(* IEC 61131-3 sources: types/src (part 3) *)

   END_TYPE

   TYPE EM480VHFDataRec145V1 : STRUCT
         version  : Byte := BYTE#1;   // Version
         resb1  : Byte;   // Reserved
         minVoltL1N  : Real;   // Min. voltage UL1-N
         minVoltL2N  : Real;   // Min. voltage UL2-N
         minVoltL3N  : Real;   // Min. voltage UL3-N
         minVoltL1L2  : Real;   // Min. voltage UL1-L2
         minVoltL2L3  : Real;   // Min. voltage UL2-L3
         minVoltL3L1  : Real;   // Min. voltage UL3-L1
         minCurrentL1  : Real;   // Min. current L1
         minCurrentL2  : Real;   // Min. current L2
         minCurrentL3  : Real;   // Min. current L3
         minApparentPowerL1  : Real;   // Min. apparent power L1
         minApparentPowerL2  : Real;   // Min. apparent power L2
         minApparentPowerL3  : Real;   // Min. apparent power L3
         minActivePowerL1  : Real;   // Min. active power L1
         minActivePowerL2  : Real;   // Min. active power L2
         minActivePowerL3  : Real;   // Min. active power L3
         minReactivePowerQtotL1  : Real;   // Min. reactive power Qtot L1
         minReactivePowerQtotL2  : Real;   // Min. reactive power Qtot L2
         minReactivePowerQtotL3  : Real;   // Min. reactive power Qtot L3
         minPowerFactorL1  : Real;   // Min. power factor L1
         minPowerFactorL2  : Real;   // Min. power factor L2
         minPowerFactorL3  : Real;   // Min. power factor L3
         minFrequency  : Real;   // Min. frequency
         minTotalApparentPower  : Real;   // Min. apparent power L1 L2 L3
         minTotalActivePower  : Real;   // Min. active power L1 L2 L3
         minTotalReactivePowerQn  : Real;   // Min. reactive power Qn L1 L2 L3
         minTotalPowerFactor  : Real;   // Min. power factor λ L1 L2 L3
         minReactivePowerQnL1  : Real;   // Min. reactive power Qn L1
         minReactivePowerQnL2  : Real;   // Min. reactive power Qn L2
         minReactivePowerQnL3  : Real;   // Min. reactive power Qn L3
         minMeanVoltLN  : Real;   // Min. mean voltage L-N
         minMeanVoltLL  : Real;   // Min. mean voltage L-L
         minTotalMeanCurr  : Real;   // Min. mean current L1 L2 L3
         minFundVoltL1  : Real;   // Min. fundamental voltage L1
         minFundVoltL2  : Real;   // Min. fundamental voltage L2
         minFundVoltL3  : Real;   // Min. fundamental voltage L3
         minFundCurrL1  : Real;   // Min. fundamental current L1
         minFundCurrL2  : Real;   // Min. fundamental current L2
         minFundCurrL3  : Real;   // Min. fundamental current L3
         minFundApparentPowerL1  : Real;   // Min. fundamental apparent power L1
         minFundApparentPowerL2  : Real;   // Min. fundamental apparent power L2
         minFundApparentPowerL3  : Real;   // Min. fundamental apparent power L3
         minFundReactivePowerL1  : Real;   // Min. fundamental reactive power L1
         minFundReactivePowerL2  : Real;   // Min. fundamental reactive power L2
         minFundReactivePowerL3  : Real;   // Min. fundamental reactive power L3
         minFundActivePowerL1  : Real;   // Min. fundamental active power L1
         minFundActivePowerL2  : Real;   // Min. fundamental active power L2
         minFundActivePowerL3  : Real;   // Min. fundamental active power L3
         minFundActiveFactorL1  : Real;   // Min. fundamental cos φ active factor L1
         minFundActiveFactorL2  : Real;   // Min. fundamental cos φ active factor L2
         minFundActiveFactorL3  : Real;   // Min. fundamental cos φ active factor L3
         minTHDaNVoltL1  : Real;   // Min. THD+N voltage L1
         minTHDaNVoltL2  : Real;   // Min. THD+N voltage L2
         minTHDaNVoltL3  : Real;   // Min. THD+N voltage L3
         minTHDaNCurrL1  : Real;   // Min. THD+N current L1
         minTHDaNCurrL2  : Real;   // Min. THD+N current L2
         minTHDaNCurrL3  : Real;   // Min. THD+N current L3
      END_STRUCT;

   END_TYPE

   TYPE EM480VHFDataRec143 : STRUCT
         version  : Byte := BYTE#1;   // Version
         resb1  : Byte;   // Reserved
         controlStatusByte1L1  : Byte;   // Status / control byte 1 - L1
         controlStatusByte2L1  : Byte;   // Status / control byte 2 - L1
         controlStatusByte1L2  : Byte;   // Status / control byte 1 - L2
         controlStatusByte2L2  : Byte;   // Status / control byte 2 - L2
         controlStatusByte1L3  : Byte;   // Status / control byte 1 - L3
         controlStatusByte2L3  : Byte;   // Status / control byte 2 - L3
         activeEnergyInLongL1  : LReal;   // Active energy inflow (initial value) L1
         activeEnergyOutLongL1  : LReal;   // Active energy outflow (initial value) L1
         reactiveEnergyInLongL1  : LReal;   // Reactive energy inflow (initial value) L1
         reactiveEnergyOutLongL1  : LReal;   // Reactive energy outflow (initial value) L1
         apparentEnergyLongL1  : LReal;   // Apparent energy (initial value) L1
         activeEnergyInLongL2  : LReal;   // Active energy inflow (initial value) L2
         activeEnergyOutLongL2  : LReal;   // Active energy outflow (initial value) L2
         reactiveEnergyInLongL2  : LReal;   // Reactive energy inflow (initial value) L2
         reactiveEnergyOutLongL2  : LReal;   // Reactive energy outflow (initial value) L2
         apparentEnergyLongL2  : LReal;   // Apparent energy (initial value) L2
         activeEnergyInLongL3  : LReal;   // Active energy inflow (initial value) L3
         activeEnergyOutLongL3  : LReal;   // Active energy outflow (initial value) L3
         reactiveEnergyInLongL3  : LReal;   // Reactive energy inflow (initial value) L3
         reactiveEnergyOutLongL3  : LReal;   // Reactive energy outflow (initial value) L3
         apparentEnergyLongL3  : LReal;   // Apparent energy (initial value) L3
         ovCntActiveEnergyInL1  : UInt;   // Overflow counter active energy inflow L1
         ovCntActiveEnergyOutL1  : UInt;   // Overflow counter active energy outflow L1
         ovCntReactiveEnergyInL1  : UInt;   // Overflow counter reactive energy inflow L1
         ovCntReactiveEnergyOutL1  : UInt;   // Overflow counter reactive energy outflow L1
         ovCntApparentEnergyL1  : UInt;   // Overflow counter apparent energy L1
         ovCntActiveEnergyInL2  : UInt;   // Overflow counter active energy inflow L2
         ovCntActiveEnergyOutL2  : UInt;   // Overflow counter active energy outflow L2
         ovCntReactiveEnergyInL2  : UInt;   // Overflow counter reactive energy inflow L2
         ovCntReactiveEnergyOutL2  : UInt;   // Overflow counter reactive energy outflow L2
         ovCntApparentEnergyL2  : UInt;   // Overflow counter apparent energy L2
         ovCntActiveEnergyInL3  : UInt;   // Overflow counter active energy inflow L3
         ovCntActiveEnergyOutL3  : UInt;   // Overflow counter active energy outflow L3
         ovCntReactiveEnergyInL3  : UInt;   // Overflow counter reactive energy inflow L3
         ovCntReactiveEnergyOutL3  : UInt;   // Overflow counter reactive energy outflow L3
         ovCntApparentEnergyL3  : UInt;   // Overflow counter apparent energy L3
         operHoursCntL1  : Real;   // Operating hours counter L1 (initial value)
         operHoursCntL2  : Real;   // Operating hours counter L2 (initial value)
         operHoursCntL3  : Real;   // Operating hours counter L2 (initial value)
      END_STRUCT;

   END_TYPE

   TYPE EM480VHFDataRec142V2 : STRUCT
         version  : Byte := BYTE#2;   // Version
         resb1  : Byte;   // Reserved
         voltL1N  : Real;   // Voltage UL1-N
         voltL2N  : Real;   // Voltage UL2-N
         voltL3N  : Real;   // Voltage UL3-N
         voltL1L2  : Real;   // Voltage UL1-L2
         voltL2L3  : Real;   // Voltage UL2-L3
         voltL3L1  : Real;   // Voltage UL3-L1
         currentL1  : Real;   // Current L1
         currentL2  : Real;   // Current L2
         currentL3  : Real;   // Current L3
         powerFactorL1  : Real;   // Power factor L1
         powerFactorL2  : Real;   // Power factor L2
         powerFactorL3  : Real;   // Power factor L3
         totalPowerFactor  : Real;   // Total power factor L1 L2 L3
         frequency  : Real;   // Frequency
         amplUnbalanceVolt  : Real;   // Amplitude unbalance for voltage
         amplUnbalanceCurrent  : Real;   // Amplitude unbalance for current
         apparentPowerL1  : Real;   // Apparent power L1
         apparentPowerL2  : Real;   // Apparent power L2
         apparentPowerL3  : Real;   // Apparent power L3
         totalApparentPower  : Real;   // Total apparent power L1 L2 L3
         reactivePowerQtotL1  : Real;   // Reactive power Qtot L1
         reactivePowerQtotL2  : Real;   // Reactive power Qtot L2
         reactivePowerQtotL3  : Real;   // Reactive power Qtot L2
         totalReactivePowerQtot  : Real;   // Total reactive power Qtot L1 L2 L3
         activePowerL1  : Real;   // Active power L1
         activePowerL2  : Real;   // Active power L2
         activePowerL3  : Real;   // Active power L3
         totalActivePower  : Real;   // Total active power L1 L2 L3
         phaseAngleL1  : Real;   //  Phase angle L1
         phaseAngleL2  : Real;   //  Phase angle L2
         phaseAngleL3  : Real;   //  Phase angle L3
         totalApparentEnergy  : Real;   // Total apparent energy L1 L2 L3
         totalReactiveEnergy  : Real;   // Total reactive energy L1 L2 L3
         totalActiveEnergy  : Real;   // Total active energy L1 L2 L3
         totalReactiveEnergyIn  : Real;   // Total reactive energy inflow L1 L2 L3
         totalReactiveEnergyOut  : Real;   // Total reactive energy outflow L1 L2 L3
         totalActiveEnergyIn  : Real;   // Total active energy inflow L1 L2 L3
         totalActiveEnergyOut  : Real;   // Total active energy outflow L1 L2 L3
         totalApparentEnergyLong  : LReal;   // Total apparent energy L1 L2 L3
         totalReactiveEnergyLong  : LReal;   // Total reactive energy L1 L2 L3
         totalActiveEnergyLong  : LReal;   // Total active energy L1 L2 L3
         totalReactiveEnergyInLong  : LReal;   // Total reactive energy inflow L1 L2 L3
         totalReactiveEnergyOutLong  : LReal;   // Total reactive energy outflow L1 L2 L3
         totalActiveEnergyInLong  : LReal;   // Total active energy inflow L1 L2 L3
         totalActiveEnergyOutLong  : LReal;   // Total active energy outflow L1 L2 L3
         neutralCurrent  : Real;   // Neutral current
      END_STRUCT;

   END_TYPE

   TYPE EM480VHFDataRec160 : STRUCT
         version  : Byte;   // Version
         resb1  : Byte;   // Reserved
         neutralCurrIn  : Real;   // Neutral current IN
         neutralCurrCyc10to12  : Real;   // Neutral current 10/12 cycles
         totalCurrIn  : Real;   // Total current IL1+IL2+IL3-IN
         totalFundReactivePower  : Real;   // Fundamental reactive power L1 L2 L3
         totalMaxFundReactivePower  : Real;   // Max. fundamental reactive power L1 L2 L3
         totalMinFundReactivePower  : Real;   // Min. fundamental reactive power L1 L2 L3
         totalPowerFactor  : Real;   // Power factor λ L1L2L3
         fundReactivePowerL1  : Real;   // Fundamental reactive power L1
         fundReactivePowerL2  : Real;   // Fundamental reactive power L2
         fundReactivePowerL3  : Real;   // Fundamental reactive power L3
         fundActiveFactorL1  : Real;   // Fundamental cos φ active factor L1
         fundActiveFactorL2  : Real;   // Fundamental cos φ active factor L2
         fundActiveFactorL3  : Real;   // Fundamental cos φ active factor L3
         THDaNVoltL1  : Real;   // THD+N voltage L1
         THDaNVoltL2  : Real;   // THD+N voltage L2
         THDaNVoltL3  : Real;   // THD+N voltage L3
         THDaNCurrL1  : Real;   // THD+N current L1
         THDaNCurrL2  : Real;   // THD+N current L2
         THDaNCurrL3  : Real;   // THD+N current L3
         maxTHDaNVoltL1  : Real;   // Max. THD+N voltage L1
         maxTHDaNVoltL2  : Real;   // Max. THD+N voltage L2
         maxTHDaNVoltL3  : Real;   // Max. THD+N voltage L3
         maxTHDaNCurrL1  : Real;   // Max. THD+N current L1
         maxTHDaNCurrL2  : Real;   // Max. THD+N current L2
         maxTHDaNCurrL3  : Real;   // Max. THD+N current L3
         minTHDaNVoltL1  : Real;   // Min. THD+N voltage L1
         minTHDaNVoltL2  : Real;   // Min. THD+N voltage L2
         minTHDaNVoltL3  : Real;   // Min. THD+N voltage L3
         minTHDaNCurrL1  : Real;   // Min. THD+N current L1
         minTHDaNCurrL2  : Real;   // Min. THD+N current L2
         minTHDaNCurrL3  : Real;   // Min. THD+N current L3
         voltDipValueL1  : Real;   // Voltage dip - value L1
         voltDipDurationL1  : Real;   // Voltage dip - duration L1
         voltDipValueL2  : Real;   // Voltage dip - value L2
         voltDipDurationL2  : Real;   // Voltage dip - duration L2
         voltDipValueL3  : Real;   // Voltage dip - value L3
         voltDipDurationL3  : Real;   // Voltage dip - duration L3
         voltIncValueL1  : Real;   // Voltage increase - value L1
         voltIncDurationL1  : Real;   // Voltage increase - duration L1
         voltIncValueL2  : Real;   // Voltage increase - value L2
         voltIncDurationL2  : Real;   // Voltage increase - duration L2
         voltIncValueL3  : Real;   // Voltage increase - value L3
         voltIncDurationL3  : Real;   // Voltage increase - duration L3
         voltPeakValueL1  : Real;   // Voltage peak value L1
         voltPeakValueL2  : Real;   // Voltage peak value L2
         voltPeakValueL3  : Real;   // Voltage peak value L3
         currPeakValueL1  : Real;   // Current peak value L1
         currPeakValueL2  : Real;   // Current peak value L2
         currPeakValueL3  : Real;   // Current peak value L3
         overCurrValueL1  : Real;   // Overcurrent value L1
         overCurrValueL2  : Real;   // Overcurrent value L2
         overCurrValueL3  : Real;   // Overcurrent value L3
         ampSymVolt  : Real;   // Amplitude symmetry Voltage U2
         ampSymCurr  : Real;   // Amplitude symmetry Current Iunsym
         powerQualityAnalysis  : UDInt;   // Power quality analysis - Qualifier
         currentModuleTime  : PNIOTimeStamp;   // Current module time
      END_STRUCT;

   END_TYPE

   TYPE EM480VHFDataRec163 : STRUCT
         version  : Byte;   // Version
         resb1  : Byte;   // Reserved
         THDaNCurrL1  : Real;   // THD+N current L1
         currL1  : Real;   // Current L1
         harmCurrL1  : Array[1..40] of Real;   // Harmonics 1-40: Current L1
         THDaNCurrL2  : Real;   // THD+N current L2
         currL2  : Real;   // Current L2
         harmCurrL2  : Array[1..40] of Real;   // Harmonics 1-40: Current L2
         THDaNCurrL3  : Real;   // THD+N current L3
         currL3  : Real;   // Current L3
         harmCurrL3  : Array[1..40] of Real;   // Harmonics 1-40: Current L3
         currentModuleTime  : PNIOTimeStamp;   // Current module time
      END_STRUCT;

   END_TYPE

   TYPE EM480VHFDataRec147V1 : STRUCT
         version  : Byte := BYTE#1;   // Version
         resb1  : Byte;   // Reserved
         qualifierL1  : Word;   // Qualifier L1
         voltL1N  : Real;   // Voltage UL1-N
         currentL1  : Real;   // Current L1
         apparentPowerL1  : Real;   // Apparent power L1
         activePowerL1  : Real;   // Active power L1
         reactivePowerL1  : Real;   // Reactive power L1
         powerFactorL1  : Real;   // Power factor L1
         phaseAngleL1  : Real;   // Phase angle L1
         apparentEnergyLongL1  : LReal;   // Apparent energy L1
         totalActiveEnergyLongL1  : LReal;   // Active energy (total) L1
         totalReactiveEnergyLongL1  : LReal;   // Reactive energy (total) L1
         maxVoltL1N  : Real;   // Max. voltage UL1-N
         maxCurrentL1  : Real;   // Max. current L1
         maxApparentPowerL1  : Real;   // Max. apparent power L1
         maxActivePowerL1  : Real;   // Max. active power L1
         maxReactivePowerL1  : Real;   // Max. reactive power L1
         maxPowerFactorL1  : Real;   // Max. power factor L1
         minVoltL1N  : Real;   // Min. voltage UL1-N
         minCurrentL1  : Real;   // Min. current L1
         minApparentPowerL1  : Real;   // Min. apparent power L1
         minActivePowerL1  : Real;   // Min. active power L1
         minReactivePowerQtotL1  : Real;   // Min. reactive power Qtot L1
         minPowerFactorL1  : Real;   // Min. power factor L1
         reactivePowerQnL1  : Real;   // Reactive power Qn L1
         voltL1Cycles10to12  : Real;   // Voltage L1 10-12 cycles
         currL1Cycles10to12  : Real;   // Current L1 10-12 cycles
         maxReactivePowerQnL1  : Real;   // Max. reactive power Qn L1
         minReactivePowerQnL1  : Real;   // Min. reactive power Qn L1
         fundVoltL1  : Real;   // Fundamental voltage L1
         fundCurrL1  : Real;   // Fundamental current L1
         fundApparentPowerL1  : Real;   // Fundamental apparent power L1
         fundReactivePowerL1  : Real;   // Fundamental reactive power L1
         fundActivePowerL1  : Real;   // Fundamental active power L1
         fundActiveFactorL1  : Real;   // Fundamental cos φ active factor L1
         maxFundVoltL1  : Real;   // Max. fundamental voltage L1
         maxFundCurrL1  : Real;   // Max. fundamental current L1
         maxFundApparentPowerL1  : Real;   // Max. fundamental apparent power L1
         maxFundReactivePowerL1  : Real;   // Max. fundamental reactive power L1
         maxFundActivePowerL1  : Real;   // Max. fundamental active power L1
         maxFundActiveFactorL1  : Real;   // Max. fundamental cos φ active factor L1
         minFundVoltL1  : Real;   // Min. fundamental voltage L1
         minFundCurrL1  : Real;   // Min. fundamental current L1
         minFundApparentPowerL1  : Real;   // Min. fundamental apparent power L1
         minFundReactivePowerL1  : Real;   // Min. fundamental reactive power L1
         minFundActivePowerL1  : Real;   // Min. fundamental active power L1
         minFundActiveFactorL1  : Real;   // Min. fundamental cos φ active factor L1
         THDaNVoltL1  : Real;   // THD+N voltage L1
         THDaNCurrL1  : Real;   // THD+N current L1
         maxTHDaNVoltL1  : Real;   // Max. THD+N voltage L1
         maxTHDaNCurrL1  : Real;   // Max. THD+N current L1
         minTHDaNVoltL1  : Real;   // Min. THD+N voltage L1
         minTHDaNCurrL1  : Real;   // Min. THD+N current L1
         voltDipValueL1  : Real;   // Voltage dip - value L1
         voltDipDurationL1  : Real;   // Voltage dip - duration L1
         voltSwellValueL1  : Real;   // Voltage swell - value L1
         voltSwellDurationL1  : Real;   // Voltage swell - duration L1
         voltPeakValueL1  : Real;   // Voltage peak value L1
         currPeakValueL1  : Real;   // Current peak value L1
         overCurrValueL1  : Real;   // Overcurrent value L1
      END_STRUCT;

   END_TYPE

   TYPE EM480VHFDataRec148V0 : STRUCT
         version  : Byte;   // Version
         resb1  : Byte;   // Reserved
         qualifierL2  : Word;   // Qualifier L2
         voltL2N  : Real;   // Voltage UL2-N
         currentL2  : Real;   // Current L2
         apparentPowerL2  : Real;   // Apparent power L2
         activePowerL2  : Real;   // Active power L2
         reactivePowerQtotL2  : Real;   // Reactive power Qtot L2
         powerFactorL2  : Real;   // Power factor L2
         phaseAngleL2  : Real;   // Phase angle L2
         apparentEnergyLongL2  : LReal;   // Apparent energy L2
         totalActiveEnergyLongL2  : LReal;   // Active energy (total) L2
         totalReactiveEnergyLongL2  : LReal;   // Reactive energy (total) L2
         maxVoltL2N  : Real;   // Max. voltage UL2-N
         maxCurrentL2  : Real;   // Max. current L2
         maxApparentPowerL2  : Real;   // Max. apparent power L2
         maxActivePowerL2  : Real;   // Max. active power L2
         maxReactivePowerQtotL2  : Real;   // Max. reactive power Qtot L2
         maxPowerFactorL2  : Real;   // Max. power factor L2
         minVoltL2N  : Real;   // Min. voltage UL2-N
         minCurrentL2  : Real;   // Min. current L2
         minApparentPowerL2  : Real;   // Min. apparent power L2
         minActivePowerL2  : Real;   // Min. active power L2
         minReactivePowerQtotL2  : Real;   // Min. reactive power L2
         minPowerFactorL2  : Real;   // Min. power factor L2
      END_STRUCT;

   END_TYPE

   TYPE EM480VHFDataRec148V1 : STRUCT
         version  : Byte := BYTE#1;   // Version
         resb1  : Byte;   // Reserved
         qualifierL2  : Word;   // Qualifier L2
         voltL2N  : Real;   // Voltage UL2-N
         currentL2  : Real;   // Current L2
         apparentPowerL2  : Real;   // Apparent power L2
         activePowerL2  : Real;   // Active power L2
         reactivePowerL2  : Real;   // Reactive power L2
         powerFactorL2  : Real;   // Power factor L2
         phaseAngleL2  : Real;   // Phase angle L2
         apparentEnergyLongL2  : LReal;   // Apparent energy L2
         totalActiveEnergyLongL2  : LReal;   // Active energy (total) L2
         totalReactiveEnergyLongL2  : LReal;   // Reactive energy (total) L2
         maxVoltL2N  : Real;   // Max. voltage UL2-N
         maxCurrentL2  : Real;   // Max. current L2
         maxApparentPowerL2  : Real;   // Max. apparent power L2
         maxActivePowerL2  : Real;   // Max. active power L2
         maxReactivePowerL2  : Real;   // Max. reactive power L2
         maxPowerFactorL2  : Real;   // Max. power factor L2
         minVoltL2N  : Real;   // Min. voltage UL2-N
         minCurrentL2  : Real;   // Min. current L2
         minApparentPowerL2  : Real;   // Min. apparent power L2
         minActivePowerL2  : Real;   // Min. active power L2
         minReactivePowerQtotL2  : Real;   // Min. reactive power Qtot L2
         minPowerFactorL2  : Real;   // Min. power factor L2
         reactivePowerQnL2  : Real;   // Reactive power Qn L2
         voltL2Cycles10to12  : Real;   // Voltage L2 10-12 cycles
         currL2Cycles10to12  : Real;   // Current L2 10-12 cycles
         maxReactivePowerQnL2  : Real;   // Max. reactive power Qn L2
         minReactivePowerQnL2  : Real;   // Min. reactive power Qn L2
         fundVoltL2  : Real;   // Fundamental voltage L2
         fundCurrL2  : Real;   // Fundamental current L2
         fundApparentPowerL2  : Real;   // Fundamental apparent power L2
         fundReactivePowerL2  : Real;   // Fundamental reactive power L2
         fundActivePowerL2  : Real;   // Fundamental active power L2
         fundActiveFactorL2  : Real;   // Fundamental cos φ active factor L2
         maxFundVoltL2  : Real;   // Max. fundamental voltage L2
         maxFundCurrL2  : Real;   // Max. fundamental current L2
         maxFundApparentPowerL2  : Real;   // Max. fundamental apparent power L2
         maxFundReactivePowerL2  : Real;   // Max. fundamental reactive power L2
         maxFundActivePowerL2  : Real;   // Max. fundamental active power L2
         maxFundActiveFactorL2  : Real;   // Max. fundamental cos φ active factor L2
         minFundVoltL2  : Real;   // Min. fundamental voltage L2
         minFundCurrL2  : Real;   // Min. fundamental current L2
         minFundApparentPowerL2  : Real;   // Min. fundamental apparent power L2
         minFundReactivePowerL2  : Real;   // Min. fundamental reactive power L2
         minFundActivePowerL2  : Real;   // Min. fundamental active power L2
         minFundActiveFactorL2  : Real;   // Min. fundamental cos φ active factor L2
         THDaNVoltL2  : Real;   // THD+N voltage L2
         THDaNCurrL2  : Real;   // THD+N current L2
         maxTHDaNVoltL2  : Real;   // Max. THD+N voltage L2
         maxTHDaNCurrL2  : Real;   // Max. THD+N current L2
         minTHDaNVoltL2  : Real;   // Min. THD+N voltage L2
         minTHDaNCurrL2  : Real;   // Min. THD+N current L2
         voltDipValueL2  : Real;   // Voltage dip - value L2
         voltDipDurationL2  : Real;   // Voltage dip - duration L2
         voltSwellValueL2  : Real;   // Voltage swell - value L2
         voltSwellDurationL2  : Real;   // Voltage swell - duration L2
         voltPeakValueL2  : Real;   // Voltage peak value L2
         currPeakValueL2  : Real;   // Current peak value L2
         overCurrValueL2  : Real;   // Overcurrent value L2
      END_STRUCT;

   END_TYPE

   TYPE EM480VHFDataRec149V0 : STRUCT
         version  : Byte;   // Version
         resb1  : Byte;   // Reserved
         qualifierL3  : Word;   // Qualifier L3
         voltL3N  : Real;   // Voltage UL3-N
         currentL3  : Real;   // Current L3
         apparentPowerL3  : Real;   // Apparent power L3
         activePowerL3  : Real;   // Active power L3
         reactivePowerQtotL3  : Real;   // Reactive power Qtot L3
         powerFactorL3  : Real;   // Power factor L3
         phaseAngleL3  : Real;   // Phase angle L3
         apparentEnergyLongL3  : LReal;   // Apparent energy L3
         totalActiveEnergyLongL3  : LReal;   // Active energy (total) L3
         totalReactiveEnergyLongL3  : LReal;   // Reactive energy (total) L3
         maxVoltL3N  : Real;   // Max. voltage UL3-N
         maxCurrentL3  : Real;   // Max. current L3
         maxApparentPowerL3  : Real;   // Max. apparent power L3
         maxActivePowerL3  : Real;   // Max. active power L3
         maxReactivePowerQtotL3  : Real;   // Max. reactive power Qtot L3
         maxPowerFactorL3  : Real;   // Max. power factor L3
         minVoltL3N  : Real;   // Min. voltage UL3-N
         minCurrentL3  : Real;   // Min. current L3
         minApparentPowerL3  : Real;   // Min. apparent power L3
         minActivePowerL3  : Real;   // Min. active power L3
         minReactivePowerQtotL3  : Real;   // Min. reactive power L3
         minPowerFactorL3  : Real;   // Min. power factor L3
      END_STRUCT;

   END_TYPE

   TYPE EM480VHFDataRec149V1 : STRUCT
         version  : Byte := BYTE#1;   // Version
         resb1  : Byte;   // Reserved
         qualifierL3  : Word;   // Qualifier L3
         voltL3N  : Real;   // Voltage UL3-N
         currentL3  : Real;   // Current L3
         apparentPowerL3  : Real;   // Apparent power L3
         activePowerL3  : Real;   // Active power L3
         reactivePowerL3  : Real;   // Reactive power L3
         powerFactorL3  : Real;   // Power factor L3
         phaseAngleL3  : Real;   // Phase angle L3
         apparentEnergyLongL3  : LReal;   // Apparent energy L3
         totalActiveEnergyLongL3  : LReal;   // Active energy (total) L3
         totalReactiveEnergyLongL3  : LReal;   // Reactive energy (total) L3
         maxVoltL3N  : Real;   // Max. voltage UL3-N
         maxCurrentL3  : Real;   // Max. current L3
         maxApparentPowerL3  : Real;   // Max. apparent power L3
         maxActivePowerL3  : Real;   // Max. active power L3
         maxReactivePowerL3  : Real;   // Max. reactive power L3
         maxPowerFactorL3  : Real;   // Max. power factor L3
         minVoltL3N  : Real;   // Min. voltage UL3-N
         minCurrentL3  : Real;   // Min. current L3
         minApparentPowerL3  : Real;   // Min. apparent power L3
         minActivePowerL3  : Real;   // Min. active power L3
         minReactivePowerQtotL3  : Real;   // Min. reactive power Qtot L3
         minPowerFactorL3  : Real;   // Min. power factor L3
         reactivePowerQnL3  : Real;   // Reactive power Qn L3
         voltL3Cycles10to12  : Real;   // Voltage L3 10-12 cycles
         currL3Cycles10to12  : Real;   // Current L3 10-12 cycles
         maxReactivePowerQnL3  : Real;   // Max. reactive power Qn L3
         minReactivePowerQnL3  : Real;   // Min. reactive power Qn L3
         fundVoltL3  : Real;   // Fundamental voltage L3
         fundCurrL3  : Real;   // Fundamental current L3
         fundApparentPowerL3  : Real;   // Fundamental apparent power L3
         fundReactivePowerL3  : Real;   // Fundamental reactive power L3
         fundActivePowerL3  : Real;   // Fundamental active power L3
         fundActiveFactorL3  : Real;   // Fundamental cos φ active factor L3
         maxFundVoltL3  : Real;   // Max. fundamental voltage L3
         maxFundCurrL3  : Real;   // Max. fundamental current L3
         maxFundApparentPowerL3  : Real;   // Max. fundamental apparent power L3
         maxFundReactivePowerL3  : Real;   // Max. fundamental reactive power L3
         maxFundActivePowerL3  : Real;   // Max. fundamental active power L3
         maxFundActiveFactorL3  : Real;   // Max. fundamental cos φ active factor L3
         minFundVoltL3  : Real;   // Min. fundamental voltage L3
         minFundCurrL3  : Real;   // Min. fundamental current L3
         minFundApparentPowerL3  : Real;   // Min. fundamental apparent power L3
         minFundReactivePowerL3  : Real;   // Min. fundamental reactive power L3
         minFundActivePowerL3  : Real;   // Min. fundamental active power L3
         minFundActiveFactorL3  : Real;   // Min. fundamental cos φ active factor L3
         THDaNVoltL3  : Real;   // THD+N voltage L3
         THDaNCurrL3  : Real;   // THD+N current L3
         maxTHDaNVoltL3  : Real;   // Max. THD+N voltage L3
         maxTHDaNCurrL3  : Real;   // Max. THD+N current L3
         minTHDaNVoltL3  : Real;   // Min. THD+N voltage L3
         minTHDaNCurrL3  : Real;   // Min. THD+N current L3
         voltDipValueL3  : Real;   // Voltage dip - value L3
         voltDipDurationL3  : Real;   // Voltage dip - duration L3
         voltSwellValueL3  : Real;   // Voltage swell - value L3
         voltSwellDurationL3  : Real;   // Voltage swell - duration L3
         voltPeakValueL3  : Real;   // Voltage peak value L3
         currPeakValueL3  : Real;   // Current peak value L3
         overCurrValueL3  : Real;   // Overcurrent value L3
      END_STRUCT;

   END_TYPE

   TYPE EM480VHFDataRec150V1 : STRUCT
         version  : Byte := BYTE#1;   // Version
         resb1  : Byte;   // Reserved
         operHoursCntTotal  : Real;   // Operating hours counter L1 L2 L3
         operHoursCntL1  : Real;   // Operating hours counter L1
         operHoursCntL2  : Real;   // Operating hours counter L2
         operHoursCntL3  : Real;   // Operating hours counter L3
         statusLimViolGW1to16  : Word;   // Status limit violation GW 1...16
         statusEnergyCntOv  : Word;   // Status of energy counter overflows
         cntLimViolGw1  : UDInt;   // Counter limit violation GW 1
         cntLimViolGw2  : UDInt;   // Counter limit violation GW 2
         cntLimViolGw3  : UDInt;   // Counter limit violation GW 3
         cntLimViolGw4  : UDInt;   // Counter limit violation GW 4
         cntLimViolGw5  : UDInt;   // Counter limit violation GW 5
         cntLimViolGw6  : UDInt;   // Counter limit violation GW 6
         cntLimViolGw7  : UDInt;   // Counter limit violation GW 7
         cntLimViolGw8  : UDInt;   // Counter limit violation GW 8
         cntLimViolGw9  : UDInt;   // Counter limit violation GW 9
         cntLimViolGw10  : UDInt;   // Counter limit violation GW 10
         cntLimViolGw11  : UDInt;   // Counter limit violation GW 11
         cntLimViolGw12  : UDInt;   // Counter limit violation GW 12
         cntLimViolGw13  : UDInt;   // Counter limit violation GW 13
         cntLimViolGw14  : UDInt;   // Counter limit violation GW 14
         cntLimViolGw15  : UDInt;   // Counter limit violation GW 15
         cntLimViolGw16  : UDInt;   // Counter limit violation GW 16
         qualifierL1L2L3  : Word;   // Qualifier L1 L2 L3
         powerQualityAnalysis  : UDInt;   // Power quality analysis - Qualifier
         currentModuleTime  : PNIOTimeStamp;   // Current module time
      END_STRUCT;

   END_TYPE

   TYPE EM480VHFDataRec151Real : STRUCT
         version  : Byte;   // Version
         numMeasValues  : Byte;   // Number of measured values for data record mapping
         measValue  : Array[1..150] of Real;   // ID of measured value for user data mapping
      END_STRUCT;

   END_TYPE

   TYPE EM480VHFDataRec161 : STRUCT
         version  : Byte;   // Version
         resb1  : Byte;   // Reserved
         THDaNVoltL1  : Real;   // THD+N voltage L1
         voltL1  : Real;   // Voltage L1
         harmVoltL1  : Array[1..40] of Real;   // Harmonics 1-40: Voltage L1
         THDaNVoltL2  : Real;   // THD+N voltage L2
         voltL2  : Real;   // Voltage L2
         harmVoltL2  : Array[1..40] of Real;   // Harmonics 1-40: Voltage L2
         THDaNVoltL3  : Real;   // THD+N voltage L3
         voltL3  : Real;   // Voltage L3
         harmVoltL3  : Array[1..40] of Real;   // Harmonics 1-40: Voltage L3
         currentModuleTime  : PNIOTimeStamp;   // Current module time
      END_STRUCT;

   END_TYPE

   TYPE EM480VHFDataRec135 : STRUCT
         majMinVer  : Byte := BYTE#0;   // Major / minor version
         dataRecordNum  : Byte := BYTE#151;   // Data record number for data record mapping = 151
         numMeasValues  : Byte := BYTE#150;   // Number of measured values for data record mapping
         resb3  : Byte;   // Reserved
         measValueID  : Array[1..150] of Word;   // ID of measured value for user data mapping
      END_STRUCT;

   END_TYPE

   TYPE TMPulseDataRec : STRUCT
         header  : TMPulseDataRecHead;   // Header
         channel  : Array[0..1] of TMPulseDataRecCh;   // Data record for 1 channel configuration; use Array[0..1] for 2 channel configuration
      END_STRUCT;

   END_TYPE

   TYPE EM480VSTDataRec130 : STRUCT
         majMinVer  : Byte := BYTE#0;   // Major / minor version
         numUserDataVariant  : Byte := BYTE#1;   // Number of user data variant = 1
         numMeasValues  : Byte;   // Number of measured values for user data mapping
         resb3  : Byte;   // Reserved
         measValue  : Array[1..64] of Word;   // ID of measured value for user data mapping
      END_STRUCT;

   END_TYPE

   TYPE EM480VSTDataRec128 : STRUCT
         majMinVer  : Byte := BYTE#81;   // Major / minor version
         numParamStruct  : Byte := BYTE#2;   // Number of parameter structures = 2
         numModuleParamBlocks  : Byte := BYTE#1;   // Number of module parameter blocks = 1
         lengthModuleParamBlock  : Byte := BYTE#8;   // Length of module parameter block = 8
         connectTypePhases  : Byte := BYTE#0;   // Connection type of the phases
         measRangePower  : Byte;   // Voltage measuring range of the power supply system
         energyCountGateScaleValLineFrequ  : Byte;   // Energy counter gate / Full-scale value for energy counter / Line frequency of the power supply system
         lineVoltTolerance  : Byte;   // Line voltage tolerance
         diagLineVolt  : Byte;   // Diagnostics line voltage
         idUserDataVariant  : Byte;   // ID of the user data variant
         resb10  : Byte;   // Reserved
         resb11  : Byte;   // Reserved
         numChannelParamBlocks  : Byte := BYTE#3;   // Number of channel parameter blocks = 3
         lengthChannelParamBlock  : Byte := BYTE#20;   // Length of channel parameter block = 20
         channel  : Array[0..2] of EM480VSTDataRecCh;
      END_STRUCT;

   END_TYPE

   TYPE MotorStarterIAndM2 : STRUCT
         blockType  : Int := 16#0022;   // Block type
         blockLength  : Int := 16#0012;   // Block length = 18
         blockVersion  : Int := 16#0100;   // Block version = 1.0
         imDate  : Array[0..15] of Char;   // Specification of an input date (YYYY-MM-DD HH:MM)
      END_STRUCT;

   END_TYPE

   TYPE MotorStarterIAndM1 : STRUCT
         blockType  : Int := 16#0021;   // Block type
         blockLength  : Int := 16#0038;   // Block length = 56
         blockVersion  : Int := 16#0100;   // Block version = 1.0
         tagFnction  : Array[0..31] of Char;   // Plant identifier
         tagLocation  : Array[0..21] of Char;   // Location designation
      END_STRUCT;

   END_TYPE

   TYPE MotorStarterIAndM0 : STRUCT
         header0  : Int;   // Reserved for header
         header2  : Int;   // Reserved for header
         header4  : Int;   // Reserved for header
         manufacturerID  : Int;   // 42 = Manufacturer ID SIEMENS
         orderID  : Array[0..19] of Char;   // Order No. (MLFB)
         serialNumber  : Array[0..15] of Char;   // Serial number
         hwRev  : Int;   // Hardware revision or product version
         swRev  : Array[0..3] of Char;   // Firmware version
         revCounter  : Int;   // Revision counter
         profileID  : Int;   // PROFIBUS profile
         profileSpecType  : Int;   // Contains further information on the profile
         imVersion  : Int;   // Version of the identification data (0101hex = Version 1.1)
         imSupported  : Int;   // Information about the available identification data (Index 2 to 4)
      END_STRUCT;

   END_TYPE

   TYPE MotorStarterDS204 : STRUCT
         blockingTime  : Byte := BYTE#2;   // Blocking time; 1 … 7,5s/0.5 s; [2 … 15]; Default [2]: 1 s.; for not safety starter mwith V1.0 t >= 5 sec [2 … 10]
         warnLimitMotorHeat  : Byte;   // Warning limit - motor heating; 0 … 99 %/1 %; [0 … 99]; [0]: Deactivated
         resw2  : Int;   // Reserved
         resw4  : Int;   // Reserved
         blockingCurrent  : Byte := BYTE#16;   // Blocking current; 150 ... 1000 %/50 %; [3 ... 20]; Default [16]: 800 %
         resb7  : Byte;   // Reserved
         lowerCurrentWarnLimit  : Byte := BYTE#7;   // Lower current warning limit; 18.75 … 100 %/3.125 %; [6 … 32]; [0]: Deactivated; Default [7]: 21.875 %
         upperCurrentWarnLimit  : Byte := BYTE#36;   // Upper current warning limit; 50 … 400 %/3.125 %; [16 … 128]; [0]: Deactivated; Default [36]: 112.5 %
      END_STRUCT;

   END_TYPE

   TYPE MotorStarterDS203 : STRUCT
         res00  : Bool;   // Reserved
         loadType  : Bool;   // Load type 0= 3phase; 1=1phase
         exMotorApp  : Bool;   // EX motor application 0= no; 1= yes (only F-Starter)
         res03  : Bool;   // Reserved
         turnOffClass0  : Bool;   // Trip class; [0]: CLASS 10; [3]: CLASS 5 (10a)
         turnOffClass1  : Bool;   // Trip class; [0]: CLASS 10; [3]: CLASS 5 (10a)
         turnOffClass2  : Bool;   // Trip class; [0]: CLASS 10; [3]: CLASS 5 (10a)
         turnOffClass3  : Bool;   // Trip class; [0]: CLASS 10; [3]: CLASS 5 (10a)
         responseOverload0  : Bool;   // Response to overload - TMM; [0]: Trip without restart; [1]: Trip with restart ; [2]: Warn only
         responseOverload1  : Bool;   // Response to overload - TMM; [0]: Trip without restart; [1]: Trip with restart ; [2]: Warn only
         behaviorThermMotorModelRestart  : Bool;   // 0]: Retention of the thermal motor; [1]: Deletion of the thermal motor
         responseSafetySwitchOff  : Bool;   // [0]: no warning by safety switch-off; [1]: warning by safety switch-off
         responseCPUStop  : Bool;   // Response to CPU STOP; [0]: Switch substitute value; [1]: Retain last value
         responseResCurrentDetect  : Bool := TRUE;   // Response to residual current; [0]: Warn ; [1]: Tripping
         responseAsymmetry  : Bool := TRUE;   // Response to asymmetry; [0]: Warn ; [1]: Tripping
         res17  : Bool;   // Reserved
         input1Level  : Bool := TRUE;   // Input 1 level; [0]: NC contact; [1]: NO contact
         input2Level  : Bool := TRUE;   // Input 2 level; [0]: NC contact; [1]: NO contact
         input3Level  : Bool := TRUE;   // Input 3 level; [0]: NC contact; [1]: NO contact
         groupFaultDiag  : Bool;   // Group fault diagnostics; [0]: Enable; [1]: Disable
         input1Signal  : Bool;   // Input 1 signal; [0]: Non-retentive; [1]: Retentive
         input2Signal  : Bool;   // Input 2 signal; [0]: Non-retentive; [1]: Retentive
         input3Signal  : Bool;   // Input 3 signal; [0]: Non-retentive; [1]: Retentive
         groupWarnDiag  : Bool := TRUE;   // Group warning diagnostics; [0]: Enable; [1]: Disable
         input1Action  : Byte := BYTE#8;   // Input 1 action; [8]: Motor CW
         input2Action  : Byte := BYTE#9;   // Input 2 action; [9]: Motor CCW
         input3Action  : Byte := BYTE#13;   // Input 3 action; [13]: Cold start; not safety starter!
         ratedOperatCurrent  : Int;   // Rated operational current Ie; 0.3 … 9 A/10 mA
         lowerCurrentLimit  : Byte;   // Lower current limit; 18.75 … 100 %/3.125 % [6 … 32]; [0]: Deactivated
         upperCurrentLimit  : Byte;   // Upper current limit; 50 … 400 %/3.125 % [16 … 128]; [0]: Deactivated
      END_STRUCT;

   END_TYPE

   TYPE MotorStarterDS95 : STRUCT
         resb0  : Byte;   // Reserved
         res10  : Bool;   // Reserved
         res11  : Bool;   // Reserved
         res12  : Bool;   // Reserved
         res13  : Bool;   // Reserved
         res14  : Bool;   // Reserved
         res15  : Bool;   // Reserved
         operatHoursResolution  : Bool;   // Operating hours resolution 1 second
         operatHoursSelect  : Bool;   // Operating hours selection 1 operating hour - device
         resw2  : Int;   // Reserved
         operatHoursDevice  : DWord;   // Device operating hours in seconds
         numStartsCw  : DInt;   // Number of motor CW starts
         numStartsCcw  : DInt;   // Number of motor CCW starts
         numOverloadTrips  : Int;   // Number of motor overload trips
         resw18  : Int;   // Reserved
         motorCurrentMax  : DInt;   // Motor current Imax; +-0...20.000A; Inc 0.01A
         lastTripCurrent  : DInt;   // Last tripping current Ia; +-0...20.000A; Inc 0.01A
         operatHoursMotor  : DInt;   // Motor operating hours in seconds
         resdw32  : DWord;   // Reserved
         resdw36  : DWord;   // Reserved
         resdw40  : DWord;   // Reserved
         resdw44  : DWord;   // Reserved
         resw48  : Word;   // Reserved
         numSwitchElemOverloadTrip  : Int;   // Number of switching element overload trips
         numHardSwitchOperatRelay  : Int;   // Number of hard switching operations of the relay
         resdw54  : DWord;   // Reserved
         resdw58  : DWord;   // Reserved
         resdw62  : DWord;   // Reserved
         resdw66  : DWord;   // Reserved
         resdw70  : DWord;   // Reserved
         resdw74  : DWord;   // Reserved
         resdw78  : DWord;   // Reserved
         resdw82  : DWord;   // Reserved
         resdw86  : DWord;   // Reserved
      END_STRUCT;

   END_TYPE

   TYPE MotorStarterDS92 : STRUCT
         ready  : Bool;   // Ready (automatic)
         motorCw  : Bool;   // Motor CW
         motorCcw  : Bool;   // Motor CCW (Reversing starters only)
         switchElementOverload  : Bool;   // Switching element overload
         switchElementDefective  : Bool;   // Switching element defective
         emergencyStartActive  : Bool;   // Emergency start active
         groupFault  : Bool;   // Group fault
         groupWarning  : Bool;   // Group warning
         res10  : Bool;   // Reserved
         res11  : Bool;   // Reserved
         res12  : Bool;   // Reserved
         res13  : Bool;   // Reserved
         res14  : Bool;   // Reserved
         res15  : Bool;   // Reserved
         res16  : Bool;   // Reserved
         res17  : Bool;   // Reserved
         res20  : Bool;   // Reserved
         res21  : Bool;   // Reserved
         res22  : Bool;   // Reserved
         thermMotorModelOverload  : Bool;   // Thermal motor model overload
         overloadTripping  : Bool;   // Overload tripping
         res25  : Bool;   // Reserved
         coolTimeActive  : Bool;   // Cooling time active
         fdiActivated  : Bool;   // Input F-DI activated (safety motor starters only)
         res30  : Bool;   // Reserved
         res31  : Bool;   // Reserved
         mechRotInterlockNotReady  : Bool;   // Mechanical rotary interlock is not in the READY position
         res33  : Bool;   // Reserved
         res34  : Bool;   // Reserved
         res35  : Bool;   // Reserved
         res36  : Bool;   // Reserved
         inputControl  : Bool;   // Input control
         asymmetryDetected  : Bool;   // Asymmetry detected
         asymmetryTripping  : Bool;   // Asymmetry tripping
         upperLimitViolation  : Bool;   // Ie upper limit violation
         lowerLimitViolation  : Bool;   // Ie lower limit violation
         res44  : Bool;   // Reserved
         residualCurrentDetected  : Bool;   // Residual current detected
         residualCurrentTripping  : Bool;   // Residual current tripping
         trippingMotorBlocking  : Bool;   // Tripping due to motor blocking
         input1  : Bool;   // Input 1
         input2  : Bool;   // Input 2
         input3  : Bool;   // Input 3
         inputLC  : Bool;   // Input LC
         inputTripping  : Bool;   // Input tripping
         inputTripCw  : Bool;   // Input trip CW
         inputWarning  : Bool;   // Input warning
         inputTripCcw  : Bool;   // Input trip CCW
         res60  : Bool;   // Reserved
         res61  : Bool;   // Reserved
         quickStopActive  : Bool;   // Quick stop active
         sensorSupplyOverload  : Bool;   // Sensor supply overload
         res64  : Bool;   // Reserved
         res65  : Bool;   // Reserved
         res66  : Bool;   // Reserved
         electSupplyVoltLow  : Bool;   // Electronics supply voltage too low
         res70  : Bool;   // Reserved
         cpuMasterStop  : Bool;   // CPU or master STOP
         autoMode  : Bool;   // Automatic mode
         res73  : Bool;   // Reserved
         manLocal  : Bool;   // Manual local (local control)
         res75  : Bool;   // Reserved
         res76  : Bool;   // Reserved
         processImageErr  : Bool;   // Process image error
         res80  : Bool;   // Reserved
         invalParaValue  : Bool;   // Invalid parameter value (during operation / starting)
         noParaChangeInOn  : Bool;   // Parameters cannot be changed in ON state
         res83  : Bool;   // Reserved
         noExtStartupParaReceiv  : Bool;   // No external startup parameters received
         res85  : Bool;   // Reserved
         res86  : Bool;   // Reserved
         res87  : Bool;   // Reserved
         res90  : Bool;   // Reserved
         res91  : Bool;   // Reserved
         faultSelfTest  : Bool;   // F-Starter: Fault self-teset
         res93  : Bool;   // Reserved
         res94  : Bool;   // Reserved
         res95  : Bool;   // Reserved
         res96  : Bool;   // Reserved
         res97  : Bool;   // Reserved
         incorrectParaNum  : Word;   // Incorrect parameter number
         resw12  : Word;   // Reserved
         coldStartActive  : Bool;   // Cold start active
         coldStartTripping  : Bool;   // Cold start tripping
         res142  : Bool;   // Reserved
         res143  : Bool;   // Reserved
         res144  : Bool;   // Reserved
         res145  : Bool;   // Reserved
         res146  : Bool;   // Reserved
         res147  : Bool;   // Reserved
         resb15  : Byte;   // Reserved
         resw16  : Word;   // Reserved
         resb18  : Byte;   // Reserved
         electSupplyVoltHigh  : Bool;   // Electronics supply voltage too high
         readyMotorOn  : Bool;   // Ready for motor ON
         switchElementShortCircuit  : Bool;   // Switching element short-circuit
         bypassElementDefect  : Bool;   // Bypass element defective
         res194  : Bool;   // Reserved
         res195  : Bool;   // Reserved
         res196  : Bool;   // Reserved
         res197  : Bool;   // Reserved
         resb20  : Byte;   // Reserved
         res210  : Bool;   // Reserved
         res211  : Bool;   // Reserved
         currMeasRangeOvershot  : Bool;   // Current measuring range overshot
         res213  : Bool;   // Reserved
         res214  : Bool;   // Reserved
         res215  : Bool;   // Reserved
         res216  : Bool;   // Reserved
         res217  : Bool;   // Reserved
         autoMode2  : Bool;   // Automatic mode (no connection to the mech. rotary interlock)
         res221  : Bool;   // Reserved
         res222  : Bool;   // Reserved
         manLocalMode  : Bool;   // Manual local mode (no connection to the mech. rotary interlock)
         res224  : Bool;   // Reserved
         res225  : Bool;   // Reserved
         res226  : Bool;   // Reserved
         res227  : Bool;   // Reserved
         resb23  : Byte;   // Reserved
         resw24  : Word;   // Reserved
         resdw26  : DWord;   // Reserved
         resw30  : Word;   // Reserved
         qickStop1Dir  : Bool;   // Quick Stop 1 - direction-independent
         qickStop1Cw  : Bool;   // Quick Stop 1 - clockwise
         qickStop1Ccw  : Bool;   // Quick Stop 1 - counter clockwise
         res323  : Bool;   // Reserved
         res324  : Bool;   // Reserved
         res325  : Bool;   // Reserved
         res326  : Bool;   // Reserved
         res327  : Bool;   // Reserved
         resb33  : Byte;   // Reserved
         endPosCw  : Bool;   // Input operational trip - end position CW
         endPosCcw  : Bool;   // Input operational trip - end position CCW
         res342  : Bool;   // Reserved
         res343  : Bool;   // Reserved
         res344  : Bool;   // Reserved
         res345  : Bool;   // Reserved
         res346  : Bool;   // Reserved
         res347  : Bool;   // Reserved
         resb35  : Byte;   // Reserved
         res360  : Bool;   // Reserved
         res361  : Bool;   // Reserved
         res362  : Bool;   // Reserved
         res363  : Bool;   // Reserved
         res364  : Bool;   // Reserved
         res365  : Bool;   // Reserved
         startPause  : Bool;   // Start_Pause command is pending
         energySaveModeActive  : Bool;   // Energy saving mode active
         resw37  : Byte;   // Reserved
         resdw38  : DWord;   // Reserved
         resdw42  : DWord;   // Reserved
         resdw46  : DWord;   // Reserved
         exMotorProtectActive  : Bool;   // F-Starter: Ex motor protection active
         res501  : Bool;   // Reserved
         newSafetyParaRec  : Bool;   // F-Starter: new safety parameters received
         res503  : Bool;   // Reserved
         res504  : Bool;   // Reserved
         res505  : Bool;   // Reserved
         res506  : Bool;   // Reserved
         res507  : Bool;   // Reserved
         resb51  : Byte;   // Reserved
         res520  : Bool;   // Reserved
         res521  : Bool;   // Reserved
         res522  : Bool;   // Reserved
         res523  : Bool;   // Reserved
         currWarnLimitExceed  : Bool;   // Ie warning limit exceeded
         currWarnLimitUndershot  : Bool;   // Ie warning limit undershot
         res526  : Bool;   // Reserved
         res527  : Bool;   // Reserved
         resb53  : Byte;   // Reserved
      END_STRUCT;

   END_TYPE

   TYPE EM480VHFDataRec129 : STRUCT
         majMinVer  : Byte := BYTE#0;   // Major / minor version
         lengthParamBlock  : Byte := BYTE#10;   // Length of parameter block = 10
         numParamBlocks  : Byte := BYTE#16;   // Number of parameter blocks
         resb3  : Byte;   // Reserved
         paramBlock  : Array[1..16] of EM480VHFDataRecParam;
      END_STRUCT;

   END_TYPE

   TYPE EM480VRCHFDataRec128 : STRUCT
         majMinVer  : Byte := BYTE#97;   // Major / minor version
         numParamStruct  : Byte := BYTE#2;   // Number of parameter structures = 2
         numModuleParamBlocks  : Byte := BYTE#1;   // Number of module parameter blocks = 1
         lengthModuleParamBlock  : Byte := BYTE#26;   // Length of module parameter block = 26
         connectTypePhases  : Byte := BYTE#0;   // Connection type of the phases
         measRangePower  : Byte;   // Voltage measuring range of the power supply system
         energyCountGateScaleValLineFrequ  : Byte;   // Energy counter gate / Full-scale value for energy counter / Line frequency of the power supply system
         resb07  : Byte;   // Reserved
         enableCalcAnalysisDiag  : Byte;   // Enable value calculation, analysis and diagnostic
         idUserDataVariant  : Byte;   // ID of the user data variant
         currTransSecVolt  : Word;   // Current transformer secondary voltage [0.1mV]
         currTransPrimCurr  : Word;   // Current transformer Primary rated current [A]
         currTransLineCond  : Byte;   // Current transformer for line conductions
         resb15  : Byte;   // Reserved
         voltDipLimit  : Word;   // Voltage dip limit in relation to nominal value voltage [0.1%]
         voltSwellLimit  : Word;   // Voltage swell limit in relation to nominal value voltage [0.1%]
         thresOverCurr  : Word;   // Threshold overcurrent in relation to nominal value current [0.1%]
         numCycForAnalysis  : Word;   // Number of cycles for analysis of voltage increase and dip
         resw24  : Word;   // Reserved
         resw26  : Word;   // Reserved
         resw28  : Word;   // Reserved
         numChannelParamBlocks  : Byte := BYTE#3;   // Number of channel parameter blocks = 3
         lengthChannelParamBlock  : Byte := BYTE#32;   // Length of channel parameter block = 32
         channel  : Array[0..2] of EM480VRCHFDataRecCh;
      END_STRUCT;

   END_TYPE

   TYPE MotorStarterIn : STRUCT
         ready : Bool;   // Ready (automatic)
         motorOn : Bool;   // Motor on
         groupFault : Bool;   // Group fault
         groupWarning : Bool;   // Group warning
         input1 : Bool;   // Input 1 (with 3DI/LC module)
         input2 : Bool;   // Input 2 (with 3DI/LC module)
         input3 : Bool;   // Input 3 (with 3DI/LC module)
         inputLC : Bool;   // Input LC (with 3DI/LC module)
         currMotorCurrentBit0 : Bool;   // Current motor current Icurr [%] Bit 0
         currMotorCurrentBit1 : Bool;   // Current motor current Icurr [%] Bit 1
         currMotorCurrentBit2 : Bool;   // Current motor current Icurr [%] Bit 2
         currMotorCurrentBit3 : Bool;   // Current motor current Icurr [%] Bit 3
         currMotorCurrentBit4 : Bool;   // Current motor current Icurr [%] Bit 4
         currMotorCurrentBit5 : Bool;   // Current motor current Icurr [%] Bit 5
         manLocalMode : Bool;   // Manual local mode (with 3DI/LC module)
         res17 : Bool;   // Reserved
         readyStartMotorOn : Bool;   // Ready to start for motor on
         motorCw : Bool;   // Motor CW
         motorCcw : Bool;   // Motor CCW (Reversing starters only)
         quickStopActive : Bool;   // Quick stop active
         energySaveModeActive : Bool;   // Energy saving mode active
         diModulePlugged : Bool;   // DI module plugged (for non safety motor starters version >= V1.1)
         exMotorProtection : Bool;   // EX motor protection (safety motor starters only)
         res27 : Bool;   // Reserved
         thermMotorModelOverload : Bool;   // Thermal motor model overload
         res31 : Bool;   // Reserved
         currentLimitTripping : Bool;   // Ie current limit tripping
         fdiActivated : Bool;   // Input F-DI activated (safety motor starters only)
         residualCurrentDetected : Bool;   // Residual current detected
         asymmetryDetected : Bool;   // Asymmetry detected
         overTemperature : Bool;   // Overtemperature
         res37 : Bool;   // Reserved
      END_STRUCT;

   END_TYPE

   TYPE EMRCHFDataRec128 : STRUCT
         majMinVer  : Byte := BYTE#105;   // Major / minor version
         numParamStruct  : Byte := BYTE#2;   // Number of parameter structures = 2
         numModuleParamBlocks  : Byte := BYTE#1;   // Number of module parameter blocks = 1
         lengthModuleParamBlock  : Byte := BYTE#26;   // Length of module parameter block = 26
         connectTypePhases  : Byte;   // Connection type of the phases
         measRangePower  : Byte;   // Voltage measuring range of the power supply system
         energyGateCountLineFrequ  : Byte;   // Energy meters gate switch / End value / Line frequency of the power supply system
         resb07  : Byte;   // Reserved
         minMaxValueCalcGateDiagVolt  : Byte;   // Min/Max value calc. / Min/Max value calc. gate / Diagnostics load voltage
         idUserDataVariant  : Byte;   // ID of the user data variant
         currTransSecVolt  : Word;   // Current transformer secondary voltage
         currTransPrimCurr  : Word;   // Current transformer primary rated current
         currTransLineCond  : Byte;   // Current transformer for line
         resb15  : Byte;   // Reserved
         voltDipLimit  : Word;   // Voltage dip limit in relation to nominal value voltage [0.1%]
         voltSwellLimit  : Word;   // Voltage swell limit in relation to nominal value voltage [0.1%]
         thresOverCurr  : Word;   // Threshold overcurrent in relation to nominal value current [0.1%]
         numCycForAnalysis  : Word;   // Number of cycles for analysis of voltage increase and dip
         resb24  : Byte;   // Reserved
         resb25  : Byte;   // Reserved
         resb26  : Byte;   // Reserved
         resb27  : Byte;   // Reserved
         resb28  : Byte;   // Reserved
         resb29  : Byte;   // Reserved
         numChannelParamBlocks  : Byte := BYTE#3;   // Number of channel parameter blocks = 3
         lengthChannelParamBlock  : Byte := BYTE#32;   // Length of channel parameter block = 32
         channel  : Array[0..2] of EMRCHFDataRecCh;   // Channels
      END_STRUCT;

   END_TYPE

   TYPE MotorStarterDS94 : STRUCT
         phaseCurrentL1  : Byte;   // Phase current L1 in %; 0...796%; Inc 3.125%
         phaseCurrentL2  : Byte;   // Phase current L2 in %; 0...796%; Inc 3.125%
         phaseCurrentL3  : Byte;   // Phase current L3 in %; 0...796%; Inc 3.125%
         resb3  : Byte;   // Reserved
         resw4  : Word;   // Reserved
         resb6  : Byte;   // Reserved
         unbalance  : Byte;   // Unbalance; 0...255%; Inc 1%
         motorHeating  : Word;   // Motor heating; 0...1.000%
         resdw10  : DWord;   // Reserved
         resdw14  : DWord;   // Reserved
         resdw18  : DWord;   // Reserved
         resdw22  : DWord;   // Reserved
         resw26  : Word;   // Reserved
         phaseCurrentEffL1  : DInt;   // Phase current L1; +-0...20.000A; Inc 0.01A
         phaseCurrentEffL2  : DInt;   // Phase current L2; +-0...20.000A; Inc 0.01A
         phaseCurrentEffL3  : DInt;   // Phase current L3; +-0...20.000A; Inc 0.01A
         electrSupplyVolt  : Int;   // Electronics supply voltage; 0... 1.500V; Inc 0.1V
         readw42  : DWord;   // Reserved
         resdw46  : DWord;   // Reserved
         resdw50  : DWord;   // Reserved
         resdw54  : DWord;   // Reserved
         resdw58  : DWord;   // Reserved
         resw62  : Word;   // Reserved
      END_STRUCT;

   END_TYPE

   TYPE MotorStarterDS7x : STRUCT
         entry : Array[1..21] of MotorStarterEntry;
      END_STRUCT;

   END_TYPE

   TYPE TMPulseControlMotor : STRUCT
         channel : Array[0..1] of TMPulseControlMotorCh;
      END_STRUCT;

   END_TYPE

   TYPE TMPulseFeedback : STRUCT
         channel : Array[0..1] of TMPulseFeedbackCh;
      END_STRUCT;

   END_TYPE

   TYPE MotorStarterIAndM3 : STRUCT
         blockType  : Int := 16#0023;   // Block type
         blockLength  : Int := 16#0038;   // Block length = 56
         blockVersion  : Int := 16#0100;   // Block version = 1.0
         imDescriptor  : Array[0..53] of Char;   // Comment
      END_STRUCT;

   END_TYPE

   TYPE EM480VSTDataRec129 : STRUCT
         majMinVer  : Byte := BYTE#0;   // Major / minor version
         lengthParamBlock  : Byte := BYTE#10;   // Length of parameter block = 10
         numParamBlocks  : Byte := BYTE#1;   // Number of parameter blocks
         resb3  : Byte;   // Reserved
         paramBlock  : Array[1..16] of EM480VSTDataRecParam;
      END_STRUCT;

   END_TYPE

   TYPE MotorStarterDS201 : STRUCT
         res00  : Bool;   // Reserved
         loadType  : Bool;   // Load type 0= 3phase; 1=1phase
         exMotorApp  : Bool;   // EX motor application 0= no; 1= yes (only F-Starter)
         res03  : Bool;   // Reserved
         turnOffClass0  : Bool;   // Trip class; [0]: CLASS 10; [3]: CLASS 5 (10a)
         turnOffClass1  : Bool;   // Trip class; [0]: CLASS 10; [3]: CLASS 5 (10a)
         turnOffClass2  : Bool;   // Trip class; [0]: CLASS 10; [3]: CLASS 5 (10a)
         turnOffClass3  : Bool;   // Trip class; [0]: CLASS 10; [3]: CLASS 5 (10a)
         responseOverload0  : Bool;   // Response to overload - TMM; [0]: Trip without restart; [1]: Trip with restart ; [2]: Warn only
         responseOverload1  : Bool;   // Response to overload - TMM; [0]: Trip without restart; [1]: Trip with restart ; [2]: Warn only
         behaviorThermMotorModelRestart  : Bool;   // 0]: Retention of the thermal motor; [1]: Deletion of the thermal motor
         responseSafetySwitchOff  : Bool;   // [0]: no warning by safety switch-off; [1]: warning by safety switch-off
         responseCPUStop  : Bool;   // Response to CPU STOP; [0]: Switch substitute value; [1]: Retain last value
         responseResCurrentDetect  : Bool := TRUE;   // Response to residual current; [0]: Warn ; [1]: Tripping
         responseAsymmetry  : Bool := TRUE;   // Response to asymmetry; [0]: Warn ; [1]: Tripping
         res17  : Bool;   // Reserved
         input1Level  : Bool := TRUE;   // Input 1 level; [0]: NC contact; [1]: NO contact
         input2Level  : Bool := TRUE;   // Input 2 level; [0]: NC contact; [1]: NO contact
         input3Level  : Bool := TRUE;   // Input 3 level; [0]: NC contact; [1]: NO contact
         groupFaultDiag  : Bool;   // Group fault diagnostics; [0]: Enable; [1]: Disable
         input1Signal  : Bool;   // Input 1 signal; [0]: Non-retentive; [1]: Retentive
         input2Signal  : Bool;   // Input 2 signal; [0]: Non-retentive; [1]: Retentive
         input3Signal  : Bool;   // Input 3 signal; [0]: Non-retentive; [1]: Retentive
         groupWarnDiag  : Bool := TRUE;   // Group warning diagnostics; [0]: Enable; [1]: Disable
         input1Action  : Byte := BYTE#8;   // Input 1 action; [8]: Motor CW
         input2Action  : Byte := BYTE#9;   // Input 2 action; [9]: Motor CCW
         input3Action  : Byte := BYTE#13;   // Input 3 action; [13]: Cold start; not safety starter!
         ratedOperatCurrent  : Int;   // Rated operational current Ie; 0.3 … 9 A/10 mA
         lowerCurrentLimit  : Byte;   // Lower current limit; 18.75 … 100 %/3.125 % [6 … 32]; [0]: Deactivated
         upperCurrentLimit  : Byte;   // Upper current limit; 50 … 400 %/3.125 % [16 … 128]; [0]: Deactivated
      END_STRUCT;

   END_TYPE

   TYPE AI2xSTDataRec128 : STRUCT
         majMinVer  : Byte := BYTE#0;   // Major / minor version
         channelParamLength  : Byte := BYTE#18;   // Length of the parameter data = 18
         channel  : Array[0..1] of AIxSTDataRecCh;
      END_STRUCT;

   END_TYPE

   TYPE EM480VCTHFDataRec128 : STRUCT
         majMinVer  : Byte := BYTE#97;   // Major / minor version
         numParamStruct  : Byte := BYTE#2;   // Number of parameter structures = 2
         numModuleParamBlocks  : Byte := BYTE#1;   // Number of module parameter blocks = 1
         lengthModuleParamBlock  : Byte := BYTE#26;   // Length of module parameter block = 26
         connectTypePhases  : Byte := BYTE#0;   // Connection type of the phases
         measRangePower  : Byte;   // Voltage measuring range of the power supply system
         energyCountGateScaleValLineFrequ  : Byte;   // Energy counter gate / Full-scale value for energy counter / Line frequency of the power supply system
         resb07  : Byte;   // Reserved
         enableCalcAnalysisDiag  : Byte;   // Enable value calculation, analysis and diagnostic
         idUserDataVariant  : Byte;   // ID of the user data variant
         currTransPrimCurr  : DWord;   // Current transformer Primary current (A)
         currTransSecCurr  : Byte;   // Current transformer secondary current; 00=1A, 01=5A
         resb15  : Byte;   // Reserved
         voltDipLimit  : Word;   // Voltage dip limit in relation to nominal value voltage [0.1%]
         voltSwellLimit  : Word;   // Voltage swell limit in relation to nominal value voltage [0.1%]
         thresOverCurr  : Word;   // Threshold overcurrent in relation to nominal value current [0.1%]
         numCycForAnalysis  : Word;   // Number of cycles for analysis of voltage increase and dip
         resw24  : Word;   // Reserved
         resw26  : Word;   // Reserved
         resw28  : Word;   // Reserved
         numChannelParamBlocks  : Byte := BYTE#3;   // Number of channel parameter blocks = 3
         lengthChannelParamBlock  : Byte := BYTE#32;   // Length of channel parameter block = 32
         channel  : Array[0..2] of EM480VCTHFDataRecCh;
      END_STRUCT;

   END_TYPE

   TYPE EM400VSTDataRec142 : STRUCT
         version  : Byte;   // Version
         resb1  : Byte;   // Reserved
         voltL1N  : Real;   // Voltage UL1-N
         voltL2N  : Real;   // Voltage UL2-N
         voltL3N  : Real;   // Voltage UL3-N
         voltL1L2  : Real;   // Voltage UL1-L2
         voltL2L3  : Real;   // Voltage UL2-L3
         voltL3L1  : Real;   // Voltage UL3-L1
         currentL1  : Real;   // Current L1
         currentL2  : Real;   // Current L2
         currentL3  : Real;   // Current L3
         powerFactorL1  : Real;   // Power factor L1
         powerFactorL2  : Real;   // Power factor L2
         powerFactorL3  : Real;   // Power factor L3
         totalPowerFactor  : Real;   // Total power factor L1 L2 L3
         frequency  : Real;   // Frequency
         amplUnbalanceVolt  : Real;   // Amplitude unbalance for voltage
         amplUnbalanceCurrent  : Real;   // Amplitude unbalance for current
         apparentPowerL1  : Real;   // Apparent power L1
         apparentPowerL2  : Real;   // Apparent power L2
         apparentPowerL3  : Real;   // Apparent power L3
         totalApparentPower  : Real;   // Total apparent power L1 L2 L3
         reactivePowerL1  : Real;   // Reactive power L1
         reactivePowerL2  : Real;   // Reactive power L2
         reactivePowerL3  : Real;   // Reactive power L2
         totalReactivePower  : Real;   // Total reactive power L1 L2 L3
         activePowerL1  : Real;   // Active power L1
         activePowerL2  : Real;   // Active power L2
         activePowerL3  : Real;   // Active power L3
         totalActivePower  : Real;   // Total active power L1 L2 L3
         phaseAngleL1  : Real;   //  Phase angle L1
         phaseAngleL2  : Real;   //  Phase angle L2
         phaseAngleL3  : Real;   //  Phase angle L3
         totalApparentEnergy  : Real;   // Total apparent energy L1 L2 L3
         totalReactiveEnergy  : Real;   // Total reactive energy L1 L2 L3
         totalActiveEnergy  : Real;   // Total active energy L1 L2 L3
         totalReactiveEnergyIn  : Real;   // Total reactive energy inflow L1 L2 L3
         totalReactiveEnergyOut  : Real;   // Total reactive energy outflow L1 L2 L3
         totalActiveEnergyIn  : Real;   // Total active energy inflow L1 L2 L3
         totalActiveEnergyOut  : Real;   // Total active energy outflow L1 L2 L3
         totalApparentEnergyLong  : LReal;   // Total apparent energy L1 L2 L3
         totalReactiveEnergyLong  : LReal;   // Total reactive energy L1 L2 L3
         totalActiveEnergyLong  : LReal;   // Total active energy L1 L2 L3
         totalReactiveEnergyInLong  : LReal;   // Total reactive energy inflow L1 L2 L3
         totalReactiveEnergyOutLong  : LReal;   // Total reactive energy outflow L1 L2 L3
         totalActiveEnergyInLong  : LReal;   // Total active energy inflow L1 L2 L3
         totalActiveEnergyOutLong  : LReal;   // Total active energy outflow L1 L2 L3
      END_STRUCT;

   END_TYPE

   TYPE EM480VHFDataRec130a131 : STRUCT
         majMinVer  : Byte := BYTE#0;   // Major / minor version
         numUserDataVariant  : Byte := BYTE#2;   // Number of user data variant = 1
         numMeasValues  : Byte := BYTE#64;   // Number of measured values for user data mapping
         resb3  : Byte;   // Reserved
         measValue  : Array[1..64] of Word;   // ID of measured value for user data mapping
      END_STRUCT;

   END_TYPE

   TYPE AI2xUIHFDataRec128V2Scale : STRUCT
         majMinVer  : Byte := BYTE#0;   // Major / minor version
         channelParamLength  : Byte := BYTE#38;   // Length of the parameter data = 38
         channel  : Array[0..1] of AI2xUIHFDataRecChV2Scale;
      END_STRUCT;

   END_TYPE

   TYPE AI4xRTDTCHFDataRec128 : STRUCT
         majMinVer  : Byte := BYTE#16;   // Major / minor version
         channelParamLength  : Byte := BYTE#22;   // Length of the parameter data = 22
         channel  : Array[0..3] of AIxRTDTCHFDataRecCh;
      END_STRUCT;

   END_TYPE

   TYPE AI4xSTDataRec128 : STRUCT
         majMinVer  : Byte := BYTE#0;   // Major / minor version
         channelParamLength  : Byte := BYTE#18;   // Length of the parameter data = 18
         channel  : Array[0..3] of AIxSTDataRecCh;
      END_STRUCT;

   END_TYPE

   TYPE AI2xUIHSDataRec128 : STRUCT
         majMinVer  : Byte := BYTE#64;   // Major / minor version
         numParamStruct  : Byte := BYTE#2;   // Number of parameter structures = 2
         numModuleParamBlocks  : Byte := BYTE#1;   // Number of module parameter blocks = 1
         lengthModuleParamBlock  : Byte := BYTE#4;   // Length of module parameter block = 4
         operatingMode  : Byte := BYTE#0;   // Operating mode
         samplingRate  : Byte;   // Sampling rate
         resw6  : Word;   // Reserved
         numChannelParamBlocks  : Byte := BYTE#2;   // Number of channel parameter blocks = 2
         lengthChannelParamBlock  : Byte := BYTE#20;   // Length of channel parameter block = 20
         channel  : Array[0..1] of AI2xUIHSDataRecCh;
      END_STRUCT;

   END_TYPE

   TYPE AI2xUIHFDataRec128V2 : STRUCT
         majMinVer  : Byte := BYTE#0;   // Major / minor version
         channelParamLength  : Byte := BYTE#22;   // Length of the parameter data = 22
         channel  : Array[0..1] of AI2xUIHFDataRecChV2;
      END_STRUCT;

   END_TYPE

   TYPE AI2xUIHFDataRec128V1 : STRUCT
         majMinVer  : Byte := BYTE#0;   // Major / minor version
         channelParamLength  : Byte := BYTE#18;   // Length of the parameter data = 18
         channel  : Array[0..1] of AI2xUIHFDataRecChV1;
      END_STRUCT;

   END_TYPE

   TYPE AI8xRTDTCHFDataRec128 : STRUCT
         majMinVer  : Byte := BYTE#16;   // Major / minor version
         channelParamLength  : Byte := BYTE#22;   // Length of the parameter data = 22
         channel  : Array[0..7] of AIxRTDTCHFDataRecCh;
      END_STRUCT;

   END_TYPE

   TYPE AI8xBADataRec128 : STRUCT
         majMinVer  : Byte := BYTE#0;   // Major / minor version
         channelParamLength  : Byte := BYTE#18;   // Length of the parameter data = 18
         channel  : Array[0..7] of AIxSTDataRecCh;
      END_STRUCT;

   END_TYPE

   TYPE AI4xIHARTDataRec140 : STRUCT
         version  : Byte := BYTE#0;   // Version
         blockLength  : Byte := BYTE#11;   // Block length = 11
         blockType  : Byte := BYTE#75;   // Block type = 75
         resb3  : Byte;   // Reserved
         variable  : Array[0..3] of AI4xIHARTDataRec140Ch;
      END_STRUCT;

   END_TYPE

   TYPE AQ2xSTDataRec128 : STRUCT
         majMinVer  : Byte := BYTE#0;   // Major / minor version
         channelParamLength  : Byte := BYTE#6;   // Length of the parameter data = 6
         channel  : Array[0..1] of AQxSTDataRecCh;
      END_STRUCT;

   END_TYPE

   TYPE AQ4xSTDataRec128 : STRUCT
         majMinVer  : Byte := BYTE#0;   // Major / minor version
         channelParamLength  : Byte := BYTE#6;   // Length of the parameter data = 6
         channel  : Array[0..3] of AQxSTDataRecCh;
      END_STRUCT;

   END_TYPE

   TYPE AI4xIHARTDataRec128 : STRUCT
         majMinVer  : Byte := BYTE#16;   // Major / minor version
         channelParamLength  : Byte := BYTE#10;   // Length of the parameter data = 10
         channel  : Array[0..3] of AI4xIHARTDataRecCh;
      END_STRUCT;

   END_TYPE

   TYPE MotorStarterDS202 : STRUCT
         blockingTime  : Byte := BYTE#2;   // Blocking time; 1 … 7,5s/0.5 s; [2 … 15]; Default [2]: 1 s.; for not safety starter mwith V1.0 t >= 5 sec [2 … 10]
         warnLimitMotorHeat  : Byte;   // Warning limit - motor heating; 0 … 99 %/1 %; [0 … 99]; [0]: Deactivated
         resw2  : Int;   // Reserved
         resw4  : Int;   // Reserved
         blockingCurrent  : Byte := BYTE#16;   // Blocking current; 150 ... 1000 %/50 %; [3 ... 20]; Default [16]: 800 %
         resb7  : Byte;   // Reserved
         lowerCurrentWarnLimit  : Byte := BYTE#7;   // Lower current warning limit; 18.75 … 100 %/3.125 %; [6 … 32]; [0]: Deactivated; Default [7]: 21.875 %
         upperCurrentWarnLimit  : Byte := BYTE#36;   // Upper current warning limit; 50 … 400 %/3.125 %; [16 … 128]; [0]: Deactivated; Default [36]: 112.5 %
      END_STRUCT;

   END_TYPE

   TYPE TMPulseControl : STRUCT
         channel : Array[0..1] of TMPulseControlCh;
      END_STRUCT;

   END_TYPE
END_NAMESPACE

(* ---- myClass.st ---- *)
NAMESPACE Simatic.Ax.Library

    {axcode:docs-v0:@simatic-ax/types:MyClass.md}
    CLASS MyClass

        VAR PUBLIC
        END_VAR

        VAR
        END_VAR

        /// Inline Comment for MyMethod. It will be shown, when you hover over the method
        /// This method has no parameters and no return value
        METHOD PUBLIC MyMethod
            ;
        END_METHOD

    END_CLASS

END_NAMESPACE
